{attribute 'qualified_only'}
VAR_GLOBAL
	visValveMaskIdx 	: UINT;
	nValveMask 			: DWORD;
	anValveMask 		: ARRAY [0..GVL_AteqConfig.nMaxProgramsToRun - 1] OF DWORD;
	nNumOfAteqDevices 	: UINT;
END_VAR

(* stored: Version 1.1.0.1
   GVL GVL_VisVariable: Id {e66e5bb2-e186-0a7a-1eb9-6daef8b222c0} *)
